{attribute 'GeneratedUsingTerminal: EP2816-0003-0016'}
{attribute addProperty BoxType "EP2816-0003-0016"}
{attribute addProperty Id "DIG_Diag_Inputs_Channel_1AT %I*DIG_Diag_Inputs_Channel_584303BF8DIG_Diag_Inputs_Channel_2AT %I*DIG_Diag_Inputs_Channel_584303BF8DIG_Inputs_DeviceAT %I*DIG_Inputs_Device_E94E5BF95DIG_Output_Channel_1AT %Q*DIG_Output_Channel_28AC1A9E8DIG_Output_Channel_2AT %Q*DIG_Output_Channel_28AC1A9E8DIG_Outputs_DeviceAT %Q*DIG_Outputs_Device_36A5EF172WcStateAT %I*WcState_9091E0EB2InfoDataAT %I*InfoData_94A18F5E2"}
{attribute addProperty CRC "2654424581"}
{attribute addProperty Size "43"}
TYPE EP2816_9E374E05 EXTENDS EtcSlaveTerminalBase_947E5A46 :
STRUCT
	{attribute addProperty Name "DIG_Diag_Inputs_Channel_1"}
	DIG_Diag_Inputs_Channel_1 : DIG_Diag_Inputs_Channel_584303BF;
	{attribute addProperty Name "DIG_Diag_Inputs_Channel_2"}
	DIG_Diag_Inputs_Channel_2 : DIG_Diag_Inputs_Channel_584303BF;
	{attribute addProperty Name "DIG_Inputs_Device"}
	DIG_Inputs_Device : DIG_Inputs_Device_E94E5BF9;
	{attribute addProperty Name "DIG_Output_Channel_1"}
	DIG_Output_Channel_1 : DIG_Output_Channel_28AC1A9E;
	{attribute addProperty Name "DIG_Output_Channel_2"}
	DIG_Output_Channel_2 : DIG_Output_Channel_28AC1A9E;
	{attribute addProperty Name "DIG_Outputs_Device"}
	DIG_Outputs_Device : DIG_Outputs_Device_36A5EF17;
	{attribute addProperty Name "WcState"}
	WcState : WcState_9091E0EB;
	{attribute addProperty Name "InfoData"}
	InfoData : InfoData_94A18F5E;
END_STRUCT
END_TYPE

(* stored: Version 1.2.0.0, ProductVersion 3.1.4024.9
   DUT EP2816_9E374E05: Id {9958f337-94d7-4d60-a275-596422b83d48} *)
